SUBAPPLICATION Uebung_249b_AX (* Asynchrone Objektattribut-Abfrage mittels gebündelter SubApp I_GetAttribute_IDA (Kommando + asynchroner Empfang in einem Baustein) bei Tasterdruck (Input_I1) und Anzeige auf OutputNumber_N1 *)
  (* Standard: 61499-2; Description: Copyright (c) 2026 Meisterschulen am Ostbahnhof This program and the accompanying materials are made available under the terms of the Eclipse Public License 2.0 which is available at https://www.eclipse.org/legal/epl-2.0/ SPDX-License-Identifier: EPL-2.0 *)
  (* Version 1.0, 2026-09-15, Franz Höpfinger, Meisterschulen am Ostbahnhof, Initial implementation of Uebung_249b_AX using I_GetAttribute_IDA SubApp *)
  PACKAGE Uebungen;
  IMPORT logiBUS::io::DI::logiBUS_DI::Input_I1;
  IMPORT Uebungen::const::UT::DefaultPool::InputNumber_I1;
  IMPORT isobus::UT::Q::const::AID::AID_IN::VALUE;
  IMPORT Uebungen::const::UT::DefaultPool_Numeric::OutputNumber_N1_N;
  IMPORT logiBUS::io::DI::logiBUS_DI_Events::BUTTON_SINGLE_CLICK;
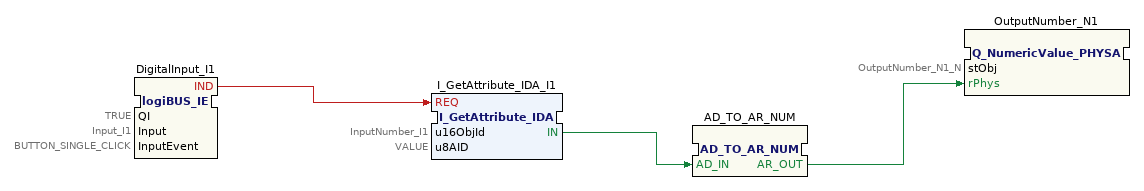
  FBS
    DigitalInput_I1 : logiBUS::io::DI::logiBUS_IE(QI := TRUE, Input := Input_I1, InputEvent := BUTTON_SINGLE_CLICK);
    AD_TO_AR_NUM : adapter::conversion::unidirectional::AD_TO_AR_NUM;
    OutputNumber_N1 : isobus::UT::Q::Q_NumericValue_PHYSA(stObj := OutputNumber_N1_N);
  END_FBS
  SUBAPPS
    I_GetAttribute_IDA_I1 : MyLib::sys::I_GetAttribute_IDA(u16ObjId := InputNumber_I1, u8AID := VALUE);
  END_SUBAPPS
  EVENT_CONNECTIONS
    DigitalInput_I1.IND TO I_GetAttribute_IDA_I1.REQ;
  END_CONNECTIONS
  ADAPTER_CONNECTIONS
    I_GetAttribute_IDA_I1.IN TO AD_TO_AR_NUM.AD_IN;
    AD_TO_AR_NUM.AR_OUT TO OutputNumber_N1.rPhys;
  END_CONNECTIONS
END_SUBAPPLICATION
